RoboDK station: palletizing_workstation.rdk

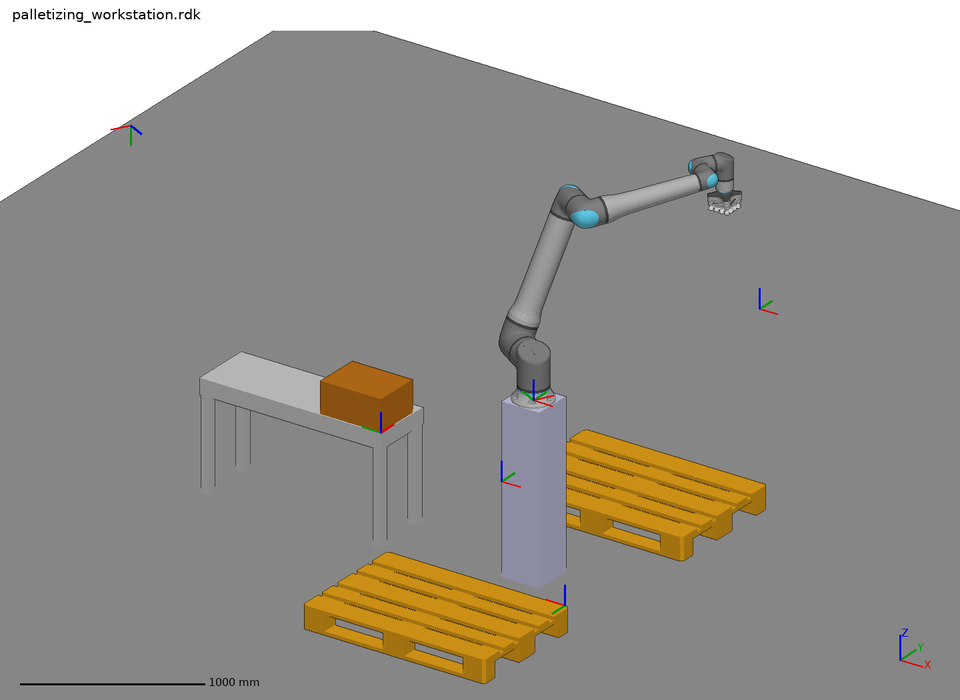
[picture v0: the station drawn from its stored meshes, robots at their saved joint values, targets as dots, program paths as lines]
Station ur_pallet (saved by RoboDK 5.7.1). Poses are relative to the parent item; angles as X-Y-Z fixed-axis rotations.
  - frame  at (0, 2128.6, 0) mm
  - frame UR20 Base at (0, 0, 300) mm
    - robot UR20: 6 axes
        modified DH rows (alpha deg, a mm, theta deg, d mm): 0, 0, 0, 236.2; 90, 0, -180, 0; 0, 861.8, 0, 0; 0, 727.7, 0, 201.9; -90, 0, 0, 159.4; 90, 0, 180, 154.8
        joint limits [-360, -360, -360, -360, -360, -360] to [360, 360, 360, 360, 360, 360]; home [0, -90, -90, 0, 90, 0]; saved at [-122.129, -68.028, 61.766, -83.74, -90.004, 147.871]
      - tool tool, TCP at (0, 0, 120) mm, size 145.3 x 145.3 x 118.3 mm
    - frame PICK_FEATURE at (-860, -211.4, -350) mm, rotated rx 0 ry 0 rz 90 deg
    - frame LEFT_PALLET_FEATURE at (-580, 528.6, -860) mm
    - frame RIGHT_PALLET_FEATURE at (580, -528.6, -860) mm, rotated rx 0 ry 0 rz 180 deg
    - frame Camera Base at (0, 0, 0) mm, rotated rx 0 ry 0 rz 62.6 deg
      - frame Camera Frame at (-280, 4158.6, -80) mm, rotated rx -90 ry 0 rz 180 deg
  - object EUR Pallet at (-590, 930, -700) mm, size 800 x 144 x 1200 mm, geometry from EUR Pallet.STEP
  - object conv at (-1360, 90, -760) mm, size 1200 x 396.3 x 703.9 mm, geometry from conv.obj
  - object EUR Pallet at (-600, -920, -700) mm, size 800 x 144 x 1200 mm, geometry from EUR Pallet.STEP
  - object base_model at (0, 0, -440) mm, size 250 x 250 x 750 mm, geometry from base_model.obj
  - object base_model at (0, 0, -750) mm, size 250 x 250 x 750 mm, geometry from base_model.obj
  - object box_0_0_0 at (-1060, -60, 150) mm, size 400 x 300 x 200 mm, geometry from box.stl
  - object box_0_0_1 at (-1060, -60, 150) mm, size 400 x 300 x 200 mm, geometry from box.stl
  - object box_0_0_2 at (-1060, -60, 150) mm, size 400 x 300 x 200 mm, geometry from box.stl
  - object box_0_0_3 at (-1060, -60, 150) mm, size 400 x 300 x 200 mm, geometry from box.stl
  - object box_0_0_4 at (-1060, -60, 150) mm, size 400 x 300 x 200 mm, geometry from box.stl
  - object box_0_0_5 at (-1060, -60, 150) mm, size 400 x 300 x 200 mm, geometry from box.stl
  - object box_0_0_6 at (-1060, -60, 150) mm, size 400 x 300 x 200 mm, geometry from box.stl
  - object box_0_0_7 at (-1060, -60, 150) mm, size 400 x 300 x 200 mm, geometry from box.stl
  - object box_0_1_0 at (-1060, -60, 150) mm, size 400 x 300 x 200 mm, geometry from box.stl
  - object box_0_1_1 at (-1060, -60, 150) mm, size 400 x 300 x 200 mm, geometry from box.stl
  - object box_0_1_2 at (-1060, -60, 150) mm, size 400 x 300 x 200 mm, geometry from box.stl
  - object box_0_1_3 at (-1060, -60, 150) mm, size 400 x 300 x 200 mm, geometry from box.stl
  - object box_0_1_4 at (-1060, -60, 150) mm, size 400 x 300 x 200 mm, geometry from box.stl
  - object box_0_1_5 at (-1060, -60, 150) mm, size 400 x 300 x 200 mm, geometry from box.stl
  - object box_0_1_6 at (-1060, -60, 150) mm, size 400 x 300 x 200 mm, geometry from box.stl
  - object box_0_1_7 at (-1060, -60, 150) mm, size 400 x 300 x 200 mm, geometry from box.stl
  - object box_0_2_0 at (-1060, -60, 150) mm, size 400 x 300 x 200 mm, geometry from box.stl
  - object box_0_2_1 at (-1060, -60, 150) mm, size 400 x 300 x 200 mm, geometry from box.stl
  - object box_0_2_2 at (-1060, -60, 150) mm, size 400 x 300 x 200 mm, geometry from box.stl
  - object box_0_2_3 at (-1060, -60, 150) mm, size 400 x 300 x 200 mm, geometry from box.stl
  - object box_0_2_4 at (-1060, -60, 150) mm, size 400 x 300 x 200 mm, geometry from box.stl
  - object box_0_2_5 at (-1060, -60, 150) mm, size 400 x 300 x 200 mm, geometry from box.stl
  - object box_0_2_6 at (-1060, -60, 150) mm, size 400 x 300 x 200 mm, geometry from box.stl
  - object box_0_2_7 at (-1060, -60, 150) mm, size 400 x 300 x 200 mm, geometry from box.stl
  - object box_0_3_0 at (-1060, -60, 150) mm, size 400 x 300 x 200 mm, geometry from box.stl
  - object box_0_3_1 at (-1060, -60, 150) mm, size 400 x 300 x 200 mm, geometry from box.stl
  - object box_0_3_2 at (-1060, -60, 150) mm, size 400 x 300 x 200 mm, geometry from box.stl
  - object box_0_3_3 at (-1060, -60, 150) mm, size 400 x 300 x 200 mm, geometry from box.stl
  - object box_0_3_4 at (-1060, -60, 150) mm, size 400 x 300 x 200 mm, geometry from box.stl
  - object box_0_3_5 at (-1060, -60, 150) mm, size 400 x 300 x 200 mm, geometry from box.stl
  - object box_0_3_6 at (-1060, -60, 150) mm, size 400 x 300 x 200 mm, geometry from box.stl
  - object box_0_3_7 at (-1060, -60, 150) mm, size 400 x 300 x 200 mm, geometry from box.stl
  - object box_1_0_0 at (-1060, -60, 150) mm, size 400 x 300 x 200 mm, geometry from box.stl
  - object box_1_0_1 at (-1060, -60, 150) mm, size 400 x 300 x 200 mm, geometry from box.stl
  - object box_1_0_2 at (-1060, -60, 150) mm, size 400 x 300 x 200 mm, geometry from box.stl
  - object box_1_0_3 at (-1060, -60, 150) mm, size 400 x 300 x 200 mm, geometry from box.stl
  - object box_1_0_4 at (-1060, -60, 150) mm, size 400 x 300 x 200 mm, geometry from box.stl
  - object box_1_0_5 at (-1060, -60, 150) mm, size 400 x 300 x 200 mm, geometry from box.stl
  - object box_1_0_6 at (-1060, -60, 150) mm, size 400 x 300 x 200 mm, geometry from box.stl
  - object box_1_0_7 at (-1060, -60, 150) mm, size 400 x 300 x 200 mm, geometry from box.stl
  - object box_1_1_0 at (-1060, -60, 150) mm, size 400 x 300 x 200 mm, geometry from box.stl
  - object box_1_1_1 at (-1060, -60, 150) mm, size 400 x 300 x 200 mm, geometry from box.stl
  - object box_1_1_2 at (-1060, -60, 150) mm, size 400 x 300 x 200 mm, geometry from box.stl
  - object box_1_1_3 at (-1060, -60, 150) mm, size 400 x 300 x 200 mm, geometry from box.stl
  - object box_1_1_4 at (-1060, -60, 150) mm, size 400 x 300 x 200 mm, geometry from box.stl
  - object box_1_1_5 at (-1060, -60, 150) mm, size 400 x 300 x 200 mm, geometry from box.stl
  - object box_1_1_6 at (-1060, -60, 150) mm, size 400 x 300 x 200 mm, geometry from box.stl
  - object box_1_1_7 at (-1060, -60, 150) mm, size 400 x 300 x 200 mm, geometry from box.stl
  - object box_1_2_0 at (-1060, -60, 150) mm, size 400 x 300 x 200 mm, geometry from box.stl
  - object box_1_2_1 at (-1060, -60, 150) mm, size 400 x 300 x 200 mm, geometry from box.stl
  - object box_1_2_2 at (-1060, -60, 150) mm, size 400 x 300 x 200 mm, geometry from box.stl
  - object box_1_2_3 at (-1060, -60, 150) mm, size 400 x 300 x 200 mm, geometry from box.stl
  - object box_1_2_4 at (-1060, -60, 150) mm, size 400 x 300 x 200 mm, geometry from box.stl
  - object box_1_2_5 at (-1060, -60, 150) mm, size 400 x 300 x 200 mm, geometry from box.stl
  - object box_1_2_6 at (-1060, -60, 150) mm, size 400 x 300 x 200 mm, geometry from box.stl
  - object box_1_2_7 at (-1060, -60, 150) mm, size 400 x 300 x 200 mm, geometry from box.stl
  - object box_1_3_0 at (-1060, -60, 150) mm, size 400 x 300 x 200 mm, geometry from box.stl
  - object box_1_3_1 at (-1060, -60, 150) mm, size 400 x 300 x 200 mm, geometry from box.stl
  - object box_1_3_2 at (-1060, -60, 150) mm, size 400 x 300 x 200 mm, geometry from box.stl
  - object box_1_3_3 at (-1060, -60, 150) mm, size 400 x 300 x 200 mm, geometry from box.stl
  - object box_1_3_4 at (-1060, -60, 150) mm, size 400 x 300 x 200 mm, geometry from box.stl
  - object box_1_3_5 at (-1060, -60, 150) mm, size 400 x 300 x 200 mm, geometry from box.stl
  - object box_1_3_6 at (-1060, -60, 150) mm, size 400 x 300 x 200 mm, geometry from box.stl
  - object box_1_3_7 at (-1060, -60, 150) mm, size 400 x 300 x 200 mm, geometry from box.stl
  - camera Camera 1
  - object floor at (0, 0, -750) mm, size 10000 x 10000 x 0 mm, geometry from floor.obj
